		MoveL Tr_meulage_bavure_P213,[50,500,0,0],z0,Tool \wobj:=Wobj_Part_0;
		MoveL Tr_meulage_bavure_P214,[50,500,0,0],z0,Tool \wobj:=Wobj_Part_0;
		MoveL Tr_meulage_bavure_P215,[50,500,0,0],z0,Tool \wobj:=Wobj_Part_0;
		MoveL Tr_meulage_bavure_P216,[50,500,0,0],z0,Tool \wobj:=Wobj_Part_0;
		MoveL Tr_meulage_bavure_P217,[50,500,0,0],z0,Tool \wobj:=Wobj_Part_0;
		MoveL Tr_meulage_bavure_P218,[50,500,0,0],z0,Tool \wobj:=Wobj_Part_0;
		MoveL Tr_meulage_bavure_P219,[50,500,0,0],z0,Tool \wobj:=Wobj_Part_0;
		MoveL Tr_meulage_bavure_P220,[50,500,0,0],z0,Tool \wobj:=Wobj_Part_0;
		MoveL Tr_meulage_bavure_P221,[50,500,0,0],z0,Tool \wobj:=Wobj_Part_0;
		MoveL Tr_meulage_bavure_P222,[50,500,0,0],z0,Tool \wobj:=Wobj_Part_0;
		MoveL Tr_meulage_bavure_P223,[50,500,0,0],z0,Tool \wobj:=Wobj_Part_0;
		MoveL Tr_meulage_bavure_P224,[50,500,0,0],z0,Tool \wobj:=Wobj_Part_0;
		MoveL Tr_meulage_bavure_P225,[50,500,0,0],z0,Tool \wobj:=Wobj_Part_0;
		MoveL Tr_meulage_bavure_P226,[50,500,0,0],z0,Tool \wobj:=Wobj_Part_0;
		MoveL Tr_meulage_bavure_P227,[50,500,0,0],z0,Tool \wobj:=Wobj_Part_0;
		MoveL Tr_meulage_bavure_P228,[50,500,0,0],z0,Tool \wobj:=Wobj_Part_0;
		MoveL Tr_meulage_bavure_P229,[50,500,0,0],z0,Tool \wobj:=Wobj_Part_0;
		MoveL Tr_meulage_bavure_P230,[50,500,0,0],z0,Tool \wobj:=Wobj_Part_0;
		MoveL Tr_meulage_bavure_P231,[50,500,0,0],z0,Tool \wobj:=Wobj_Part_0;
		MoveL Tr_meulage_bavure_P232,[50,500,0,0],z0,Tool \wobj:=Wobj_Part_0;
		MoveL Tr_meulage_bavure_P233,[50,500,0,0],z0,Tool \wobj:=Wobj_Part_0;
		MoveL Tr_meulage_bavure_P234,[50,500,0,0],z0,Tool \wobj:=Wobj_Part_0;
		MoveL Tr_meulage_bavure_P235,[50,500,0,0],z0,Tool \wobj:=Wobj_Part_0;
		MoveL Tr_meulage_bavure_P236,[50,500,0,0],z0,Tool \wobj:=Wobj_Part_0;
		MoveL Tr_meulage_bavure_P237,[50,500,0,0],z0,Tool \wobj:=Wobj_Part_0;
		MoveL Tr_meulage_bavure_P238,[50,500,0,0],z0,Tool \wobj:=Wobj_Part_0;
		MoveL Tr_meulage_bavure_P239,[50,500,0,0],z0,Tool \wobj:=Wobj_Part_0;
		MoveL Tr_meulage_bavure_P240,[50,500,0,0],z0,Tool \wobj:=Wobj_Part_0;
		MoveL Tr_meulage_bavure_P241,[50,500,0,0],z0,Tool \wobj:=Wobj_Part_0;
		MoveL Tr_meulage_bavure_P242,[50,500,0,0],z0,Tool \wobj:=Wobj_Part_0;
		MoveL Tr_meulage_bavure_P243,[50,500,0,0],z0,Tool \wobj:=Wobj_Part_0;
		MoveL Tr_meulage_bavure_P244,[50,500,0,0],z0,Tool \wobj:=Wobj_Part_0;
		MoveL Tr_meulage_bavure_P245,[50,500,0,0],z0,Tool \wobj:=Wobj_Part_0;
		MoveL Tr_meulage_bavure_P246,[50,500,0,0],z0,Tool \wobj:=Wobj_Part_0;
		MoveL Tr_meulage_bavure_P247,[50,500,0,0],z0,Tool \wobj:=Wobj_Part_0;
		MoveL Tr_meulage_bavure_P248,[50,500,0,0],z0,Tool \wobj:=Wobj_Part_0;
		MoveL Tr_meulage_bavure_P249,[50,500,0,0],z0,Tool \wobj:=Wobj_Part_0;
		MoveL Tr_meulage_bavure_P250,[50,500,0,0],z0,Tool \wobj:=Wobj_Part_0;
		MoveL Tr_meulage_bavure_P251,[50,500,0,0],z0,Tool \wobj:=Wobj_Part_0;
		MoveL Tr_meulage_bavure_P252,[50,500,0,0],z0,Tool \wobj:=Wobj_Part_0;
		MoveL Tr_meulage_bavure_P253,[50,500,0,0],z0,Tool \wobj:=Wobj_Part_0;
		MoveL Tr_meulage_bavure_P254,[50,500,0,0],z0,Tool \wobj:=Wobj_Part_0;
		MoveL Tr_meulage_bavure_P255,[50,500,0,0],z0,Tool \wobj:=Wobj_Part_0;
		MoveL Tr_meulage_bavure_P256,[50,500,0,0],z0,Tool \wobj:=Wobj_Part_0;
		MoveL Tr_meulage_bavure_P257,[50,500,0,0],z0,Tool \wobj:=Wobj_Part_0;
		MoveL Tr_meulage_bavure_P258,[50,500,0,0],z0,Tool \wobj:=Wobj_Part_0;
		MoveL Tr_meulage_bavure_P259,[50,500,0,0],z0,Tool \wobj:=Wobj_Part_0;
		MoveL Tr_meulage_bavure_P260,[50,500,0,0],z0,Tool \wobj:=Wobj_Part_0;
		MoveL Tr_meulage_bavure_P261,[50,500,0,0],z0,Tool \wobj:=Wobj_Part_0;
		MoveL Tr_meulage_bavure_P262,[50,500,0,0],z0,Tool \wobj:=Wobj_Part_0;
		MoveL Tr_meulage_bavure_P263,[50,500,0,0],z0,Tool \wobj:=Wobj_Part_0;
		MoveL Tr_meulage_bavure_P264,[50,500,0,0],z0,Tool \wobj:=Wobj_Part_0;
		MoveL Tr_meulage_bavure_P265,[50,500,0,0],z0,Tool \wobj:=Wobj_Part_0;
		MoveL Tr_meulage_bavure_P266,[50,500,0,0],z0,Tool \wobj:=Wobj_Part_0;
		MoveL Tr_meulage_bavure_P267,[50,500,0,0],z0,Tool \wobj:=Wobj_Part_0;
		MoveL Tr_meulage_bavure_P268,[50,500,0,0],z0,Tool \wobj:=Wobj_Part_0;
		MoveL Tr_meulage_bavure_P269,[50,500,0,0],z0,Tool \wobj:=Wobj_Part_0;
		MoveL Tr_meulage_bavure_P270,[50,500,0,0],z0,Tool \wobj:=Wobj_Part_0;
		MoveL Tr_meulage_bavure_P271,[50,500,0,0],z0,Tool \wobj:=Wobj_Part_0;
		MoveL Tr_meulage_bavure_P272,[50,500,0,0],z0,Tool \wobj:=Wobj_Part_0;
		MoveL Tr_meulage_bavure_P273,[50,500,0,0],z0,Tool \wobj:=Wobj_Part_0;
		MoveL Tr_meulage_bavure_P274,[50,500,0,0],z0,Tool \wobj:=Wobj_Part_0;
		MoveL Tr_meulage_bavure_P275,[50,500,0,0],z0,Tool \wobj:=Wobj_Part_0;
		MoveL Tr_meulage_bavure_P276,[50,500,0,0],z0,Tool \wobj:=Wobj_Part_0;
		MoveL Tr_meulage_bavure_P277,[50,500,0,0],z0,Tool \wobj:=Wobj_Part_0;
		MoveL Tr_meulage_bavure_P278,[50,500,0,0],z0,Tool \wobj:=Wobj_Part_0;
		MoveL Tr_meulage_bavure_P279,[50,500,0,0],z0,Tool \wobj:=Wobj_Part_0;
		MoveL Tr_meulage_bavure_P280,[50,500,0,0],z0,Tool \wobj:=Wobj_Part_0;
		MoveL Tr_meulage_bavure_P281,[50,500,0,0],z0,Tool \wobj:=Wobj_Part_0;
		MoveL Tr_meulage_bavure_P282,[50,500,0,0],z0,Tool \wobj:=Wobj_Part_0;
		MoveL Tr_meulage_bavure_P283,[50,500,0,0],z0,Tool \wobj:=Wobj_Part_0;
		MoveL Tr_meulage_bavure_P284,[50,500,0,0],z0,Tool \wobj:=Wobj_Part_0;
		MoveL Tr_meulage_bavure_P285,[50,500,0,0],z0,Tool \wobj:=Wobj_Part_0;
		MoveL Tr_meulage_bavure_P286,[50,500,0,0],z0,Tool \wobj:=Wobj_Part_0;
		MoveL Tr_meulage_bavure_P287,[50,500,0,0],z0,Tool \wobj:=Wobj_Part_0;
		MoveL Tr_meulage_bavure_P288,[50,500,0,0],z0,Tool \wobj:=Wobj_Part_0;
		MoveL Tr_meulage_bavure_P289,[50,500,0,0],z0,Tool \wobj:=Wobj_Part_0;
		MoveL Tr_meulage_bavure_P290,[50,500,0,0],z0,Tool \wobj:=Wobj_Part_0;
		MoveL Tr_meulage_bavure_P291,[50,500,0,0],z0,Tool \wobj:=Wobj_Part_0;
		MoveL Tr_meulage_bavure_P292,[50,500,0,0],z0,Tool \wobj:=Wobj_Part_0;
		MoveL Tr_meulage_bavure_P293,[50,500,0,0],z0,Tool \wobj:=Wobj_Part_0;
		MoveL Tr_meulage_bavure_P294,[50,500,0,0],z0,Tool \wobj:=Wobj_Part_0;
		MoveL Tr_meulage_bavure_P295,[50,500,0,0],z0,Tool \wobj:=Wobj_Part_0;
		MoveL Tr_meulage_bavure_P296,[50,500,0,0],z0,Tool \wobj:=Wobj_Part_0;
		MoveL Tr_meulage_bavure_P297,[50,500,0,0],z0,Tool \wobj:=Wobj_Part_0;
		MoveL Tr_meulage_bavure_P298,[50,500,0,0],z0,Tool \wobj:=Wobj_Part_0;
		MoveL Tr_meulage_bavure_P299,[50,500,0,0],z0,Tool \wobj:=Wobj_Part_0;
		MoveL Tr_meulage_bavure_P300,[50,500,0,0],z0,Tool \wobj:=Wobj_Part_0;
		MoveL Tr_meulage_bavure_P301,[50,500,0,0],z0,Tool \wobj:=Wobj_Part_0;
		MoveL Tr_meulage_bavure_P302,[50,500,0,0],z0,Tool \wobj:=Wobj_Part_0;
		MoveL Tr_meulage_bavure_P303,[50,500,0,0],z0,Tool \wobj:=Wobj_Part_0;
		MoveL Tr_meulage_bavure_P304,[50,500,0,0],z0,Tool \wobj:=Wobj_Part_0;
		MoveL Tr_meulage_bavure_P305,[50,500,0,0],z0,Tool \wobj:=Wobj_Part_0;
		MoveL Tr_meulage_bavure_P306,[50,500,0,0],z0,Tool \wobj:=Wobj_Part_0;
		MoveL Tr_meulage_bavure_P307,[50,500,0,0],z0,Tool \wobj:=Wobj_Part_0;
		MoveL Tr_meulage_bavure_P308,[50,500,0,0],z0,Tool \wobj:=Wobj_Part_0;
		MoveL Tr_meulage_bavure_P309,[50,500,0,0],z0,Tool \wobj:=Wobj_Part_0;
		MoveL Tr_meulage_bavure_P310,[50,500,0,0],z0,Tool \wobj:=Wobj_Part_0;
		MoveL Tr_meulage_bavure_P311,[50,500,0,0],z0,Tool \wobj:=Wobj_Part_0;
		MoveL Tr_meulage_bavure_P312,[50,500,0,0],z0,Tool \wobj:=Wobj_Part_0;
		MoveL Tr_meulage_bavure_P313,[50,500,0,0],z0,Tool \wobj:=Wobj_Part_0;
		MoveL Tr_meulage_bavure_P314,[50,500,0,0],z0,Tool \wobj:=Wobj_Part_0;
		MoveL Tr_meulage_bavure_P315,[50,500,0,0],z0,Tool \wobj:=Wobj_Part_0;
		MoveL Tr_meulage_bavure_P316,[50,500,0,0],z0,Tool \wobj:=Wobj_Part_0;
		MoveL Tr_meulage_bavure_P317,[50,500,0,0],z0,Tool \wobj:=Wobj_Part_0;
		MoveL Tr_meulage_bavure_P318,[50,500,0,0],z0,Tool \wobj:=Wobj_Part_0;
		MoveL Tr_meulage_bavure_P319,[50,500,0,0],z0,Tool \wobj:=Wobj_Part_0;
		MoveL Tr_meulage_bavure_P320,[50,500,0,0],z0,Tool \wobj:=Wobj_Part_0;
		MoveL Tr_meulage_bavure_P321,[50,500,0,0],z0,Tool \wobj:=Wobj_Part_0;
		MoveL Tr_meulage_bavure_P322,[50,500,0,0],z0,Tool \wobj:=Wobj_Part_0;
		MoveL Tr_meulage_bavure_P323,[50,500,0,0],z0,Tool \wobj:=Wobj_Part_0;
		MoveL Tr_meulage_bavure_P324,[50,500,0,0],z0,Tool \wobj:=Wobj_Part_0;
		MoveL Tr_meulage_bavure_P325,[50,500,0,0],z0,Tool \wobj:=Wobj_Part_0;
		MoveL Tr_meulage_bavure_P326,[50,500,0,0],z0,Tool \wobj:=Wobj_Part_0;
		MoveL Tr_meulage_bavure_P327,[50,500,0,0],z0,Tool \wobj:=Wobj_Part_0;
		MoveL Tr_meulage_bavure_P328,[50,500,0,0],z0,Tool \wobj:=Wobj_Part_0;
		MoveL Tr_meulage_bavure_P329,[50,500,0,0],z0,Tool \wobj:=Wobj_Part_0;
		MoveL Tr_meulage_bavure_P330,[50,500,0,0],z0,Tool \wobj:=Wobj_Part_0;
		MoveL Tr_meulage_bavure_P331,[50,500,0,0],z0,Tool \wobj:=Wobj_Part_0;
		MoveL Tr_meulage_bavure_P332,[50,500,0,0],z0,Tool \wobj:=Wobj_Part_0;
		MoveL Tr_meulage_bavure_P333,[50,500,0,0],z0,Tool \wobj:=Wobj_Part_0;
		MoveL Tr_meulage_bavure_P334,[50,500,0,0],z0,Tool \wobj:=Wobj_Part_0;
		MoveL Tr_meulage_bavure_P335,[50,500,0,0],z0,Tool \wobj:=Wobj_Part_0;
		MoveL Tr_meulage_bavure_P336,[50,500,0,0],z0,Tool \wobj:=Wobj_Part_0;
		MoveL Tr_meulage_bavure_P337,[50,500,0,0],z0,Tool \wobj:=Wobj_Part_0;
		MoveL Tr_meulage_bavure_P338,[50,500,0,0],z0,Tool \wobj:=Wobj_Part_0;
		MoveL Tr_meulage_bavure_P339,[50,500,0,0],z0,Tool \wobj:=Wobj_Part_0;
		MoveL Tr_meulage_bavure_P340,[50,500,0,0],z0,Tool \wobj:=Wobj_Part_0;
		MoveL Tr_meulage_bavure_P341,[50,500,0,0],z0,Tool \wobj:=Wobj_Part_0;
		MoveL Tr_meulage_bavure_P342,[50,500,0,0],z0,Tool \wobj:=Wobj_Part_0;
		MoveL Tr_meulage_bavure_P343,[50,500,0,0],z0,Tool \wobj:=Wobj_Part_0;
		MoveJ Tr_meulage_bavure_degg1,V500,Z0,Tool,\Wobj:=Wobj_Part_0;
		MoveJ Tr_meulage_bavure_degg2,V2000,Z100,Tool,\Wobj:=Wobj_Part_0;
	ENDPROC
	 PROC P36_MAIN()
		Tr_pick;
		Tr_Cut;
		Tr_meulage_motif_1;
		Tr_meulage_motif_2;
		Tr_meulage_bavure;
	ENDPROC
ENDMODULE
